VAR_GLOBAL
    KommAnVisu                 : INT;      (* Kommunikation an die Visualisierung *)
    KommVonVisu                : INT;      (* Kommunikation von der Visualisierung *)
    belegt                     : BOOL;     (* true = erzeugt Dummyteil, false = keine Auswirkungen (nur Handauflage) *)
    daten_gebucht              : BOOL;
    SteuerStatus               : DUT_Visu_SteuerStatus;

    // Frequenzumrichter
    //transport                : DUT_SEW_FU_Visu;       //#Tab:  #Name: 

    // Servoregler
    //Achse                    : DUT_Achse_Service;      //#Tab: #Name: 

    // Ventile
	 Niederhalter        		: DUT_Ventil_VISU;      //#Tab: 3530 Transport #Name: Schlossseite Längsanschlag

END_VAR

VAR_GLOBAL PERSISTENT
    Schrittnummer           : INT;
    Kopfdaten               : DUT_Kopfdaten;
    Kopfdaten_default       : DUT_Kopfdaten;
    Jobdaten                : ARRAY[1..GVL_3000.cSize_Jobdaten] OF DUT_Jobdaten;
    Jobdaten_default        : ARRAY[1..GVL_3000.cSize_Jobdaten] OF DUT_Jobdaten;
	aktJob					: DUT_Jobdaten;
	iJobNr					: INT := 1;

    //para_Vorlage             : REAL := 0.0; //#Typ: VParam #Tab:  #Name:  #Einheit:mm #Min: 1 #Max: 100 #Format:F1
END_VAR

(* stored: Version 1.1.0.1
   GVL GVL_Visu_3530: Id {578ac80b-0a4c-4dcc-b366-25ffca4c81f9} *)
